(*

## Short summary
This class provides assert statements for pointers  

.. <legal notes>

legal notes
=================
| SPDX-FileCopyrightText: © 2022 ekvip automation GmbH <info@ekvip.de>
| SPDX-License-Identifier: Apache-2.0
| For details check: Apache-2.0_

.. _Apache-2.0: https://www.apache.org/licenses/LICENSE-2.0

.. </legal notes>



*)

{attribute 'reflection'}
FUNCTION_BLOCK PointerAssertions EXTENDS AbstractAssertion IMPLEMENTS IPointerAssertions
VAR
END_VAR

(*

## Short summary
This abstract property returns the class name of the concrete object, 
It's for debugging purpose

.. <legal notes>

legal notes
=================
| SPDX-FileCopyrightText: © 2022 ekvip automation GmbH <info@ekvip.de>
| SPDX-License-Identifier: Apache-2.0
| For details check: Apache-2.0_

.. _Apache-2.0: https://www.apache.org/licenses/LICENSE-2.0

.. </legal notes>

*)

PROPERTY className :CNM_AbstractObject.ClassName
GET
className := 'CNM_Assertor.PointerAssertions';
END_GET
END_PROPERTY

(*

## Short summary
This assertion method checks if pointer is aligned with register size.

.. <legal notes>

legal notes
=================
| SPDX-FileCopyrightText: © 2025 ekvip automation GmbH <info@ekvip.de>
| SPDX-License-Identifier: Apache-2.0
| For details check: Apache-2.0_

.. _Apache-2.0: https://www.apache.org/licenses/LICENSE-2.0

.. </legal notes>



*)

METHOD isAligned
VAR_INPUT
	(* memory address *)
	address		:PVOID;
	(* message if the assertion is false *)
	message		:AssertMessage;
END_VAR
VAR CONSTANT
	SIZE :PVOID := SIZEOF(__XWORD);
END_VAR
IF (address MOD SIZE > 0) THEN
	THIS^.assertionWasWrong(message, THIS^.getDebugInfo('isAligned'));
END_IF
END_METHOD

(*

## Short summary
This assertion method checks if pointer is aligned with DWord size.

.. <legal notes>

legal notes
=================
| SPDX-FileCopyrightText: © 2025 ekvip automation GmbH <info@ekvip.de>
| SPDX-License-Identifier: Apache-2.0
| For details check: Apache-2.0_

.. _Apache-2.0: https://www.apache.org/licenses/LICENSE-2.0

.. </legal notes>



*)

METHOD isDwordAligned
VAR_INPUT
	(* memory address *)
	address		:PVOID;
	(* message if the assertion is false *)
	message		:AssertMessage;
END_VAR
VAR CONSTANT
	SIZE :PVOID := SIZEOF(DWORD);
END_VAR
IF (address MOD SIZE > 0) THEN
	THIS^.assertionWasWrong(message, THIS^.getDebugInfo('isAligned'));
END_IF
END_METHOD

(*

## Short summary
This assertion method checks if ``address1`` and ``address2`` refer to the same address

.. <legal notes>

legal notes
=================
| SPDX-FileCopyrightText: © 2022 ekvip automation GmbH <info@ekvip.de>
| SPDX-License-Identifier: Apache-2.0
| For details check: Apache-2.0_

.. _Apache-2.0: https://www.apache.org/licenses/LICENSE-2.0

.. </legal notes>



*)

METHOD isEqualTo
VAR_INPUT
	(* memory address *)
	address1	:PVOID;
	(* memory address *)
	address2	:PVOID;
	(* message if the assertion is false *)
	message		:AssertMessage;
END_VAR
IF (address1 <> address2) THEN
	THIS^.assertionWasWrong(message, THIS^.getDebugInfo('isEqualTo'));
END_IF
END_METHOD

(*

## Short summary
This assertion method checks if pointer is aligned with Lword size.

.. <legal notes>

legal notes
=================
| SPDX-FileCopyrightText: © 2025 ekvip automation GmbH <info@ekvip.de>
| SPDX-License-Identifier: Apache-2.0
| For details check: Apache-2.0_

.. _Apache-2.0: https://www.apache.org/licenses/LICENSE-2.0

.. </legal notes>



*)

METHOD isLwordAligned
VAR_INPUT
	(* memory address *)
	address		:PVOID;
	(* message if the assertion is false *)
	message		:AssertMessage;
END_VAR
VAR CONSTANT
	SIZE :PVOID := SIZEOF(LWORD);
END_VAR
IF (address MOD SIZE > 0) THEN
	THIS^.assertionWasWrong(message, THIS^.getDebugInfo('isAligned'));
END_IF
END_METHOD

(*

## Short summary
This assertion method checks if ``address1`` and ``address2`` refer not to the same address

.. <legal notes>

legal notes
=================
| SPDX-FileCopyrightText: © 2022 ekvip automation GmbH <info@ekvip.de>
| SPDX-License-Identifier: Apache-2.0
| For details check: Apache-2.0_

.. _Apache-2.0: https://www.apache.org/licenses/LICENSE-2.0

.. </legal notes>



*)

METHOD isNotEqualTo
VAR_INPUT
	(* memory address *)
	address1	:PVOID;
	(* memory address *)
	address2	:PVOID;
	(* message if the assertion is false *)
	message		:AssertMessage;
END_VAR
IF (address1 = address2) THEN
	THIS^.assertionWasWrong(message, THIS^.getDebugInfo('isNotEqualTo'));
END_IF
END_METHOD

(*

## Short summary
This assertion method checks if pointer is not null

.. <legal notes>

legal notes
=================
| SPDX-FileCopyrightText: © 2022 ekvip automation GmbH <info@ekvip.de>
| SPDX-License-Identifier: Apache-2.0
| For details check: Apache-2.0_

.. _Apache-2.0: https://www.apache.org/licenses/LICENSE-2.0

.. </legal notes>



*)

METHOD isNotNull
VAR_INPUT
	(* memory address *)
	address	:PVOID;
	(* message if the assertion is false *)
	message	:AssertMessage;
END_VAR
IF (address = 0) THEN
	THIS^.assertionWasWrong(message, THIS^.getDebugInfo('isNotNull'));
END_IF
END_METHOD

(*

## Short summary
This assertion method checks if memory areas are overlapping

.. <legal notes>

legal notes
=================
| SPDX-FileCopyrightText: © 2022 ekvip automation GmbH <info@ekvip.de>
| SPDX-License-Identifier: Apache-2.0
| For details check: Apache-2.0_

.. _Apache-2.0: https://www.apache.org/licenses/LICENSE-2.0

.. </legal notes>



*)

METHOD isNotOverlapping
VAR_INPUT
	(* memory address *)
	address1	:PVOID;
	(* memory address *)
	address2	:PVOID;
	(*the size of the memory area identified by address1*)
	sizeInBytes1		:UDINT;
	(*the size of the memory area identified by address2*)
	sizeInBytes2		:UDINT;
	(* message if the assertion is false *)
	message		:AssertMessage;
END_VAR
IF 	(( 
		address1 = address2
	) OR_ELSE(
		//address1 + sizeInBytes1 < address1 is to protect overflows caused by the calculation address1 + sizeInBytes1
		(address1 < address2) AND_THEN ((address1 + sizeInBytes1 < address1) OR_ELSE ((address1 + sizeInBytes1) >= address2))
	) OR_ELSE (
		//address2 + sizeInBytes2 < address2 is to protect overflows caused by the calculation address2 + sizeInBytes2
		(address1 > address2) AND_THEN (((address2 + sizeInBytes2 < address2) OR_ELSE ((address2 + sizeInBytes2) >= address1)))
	)
) THEN
		THIS^.assertionWasWrong(message, THIS^.getDebugInfo('isNotOverlapping'));
END_IF
END_METHOD

(*

## Short summary
This assertion method checks if pointer is null

.. <legal notes>

legal notes
=================
| SPDX-FileCopyrightText: © 2022 ekvip automation GmbH <info@ekvip.de>
| SPDX-License-Identifier: Apache-2.0
| For details check: Apache-2.0_

.. _Apache-2.0: https://www.apache.org/licenses/LICENSE-2.0

.. </legal notes>



*)

METHOD isNull
VAR_INPUT
	(* memory address *)
	address	:PVOID;
	(* message if the assertion is false *)
	message	:AssertMessage;
END_VAR
IF (address <> 0) THEN
	THIS^.assertionWasWrong(message, THIS^.getDebugInfo('isNull'));
END_IF
END_METHOD

(*

## Short summary
This assertion method checks if memory areas are overlapping

.. <legal notes>

legal notes
=================
| SPDX-FileCopyrightText: © 2022 ekvip automation GmbH <info@ekvip.de>
| SPDX-License-Identifier: Apache-2.0
| For details check: Apache-2.0_

.. _Apache-2.0: https://www.apache.org/licenses/LICENSE-2.0

.. </legal notes>



*)

METHOD isOverlapping
VAR_INPUT
	(* memory address *)
	address1	:PVOID;
	(* memory address *)
	address2	:PVOID;
	(*the size of the memory area identified by address1*)
	sizeInBytes1		:UDINT;
	(*the size of the memory area identified by address2*)
	sizeInBytes2		:UDINT;
	(* message if the assertion is false *)
	message		:AssertMessage;
END_VAR
RETURN(address1 = address2);
IF ((
		(address1 < address2) AND_THEN ((address1 + sizeInBytes1) < address2)
	) OR_ELSE (
		(address1 > address2) AND_THEN ((address2 + sizeInBytes2) < address1)
	)
) THEN
	THIS^.assertionWasWrong(message, THIS^.getDebugInfo('isOverlapping'));
END_IF;
END_METHOD

(*

## Short summary
This assertion method checks if pointer is valid.
That means the pointer and size are not zero,
the pointer is in a valid area.

**Attention:** 
	Validity of the pointer will be proofed for 32 bit systems only.
	For other systems it's an optimistic estimate.

.. <legal notes>

legal notes
=================
| SPDX-FileCopyrightText: © 2022 ekvip automation GmbH <info@ekvip.de>
| SPDX-License-Identifier: Apache-2.0
| For details check: Apache-2.0_

.. _Apache-2.0: https://www.apache.org/licenses/LICENSE-2.0

.. </legal notes>



*)

METHOD isValid
VAR_INPUT
	(* memory address *)
	address		:PVOID;
	(* number of bytes *)
	sizeInBytes	:UDINT;
	(* message if the assertion is false *)
	message		:AssertMessage;
END_VAR
VAR
	{attribute 'displaymode':='hex'}
	stackAddress	:__XWORD;
	testPointer		:POINTER TO BYTE := NULL;
	testByte		:BYTE;
	exc				: __SYSTEM.ExceptionCode;
END_VAR
VAR CONSTANT
	{attribute 'displaymode':='hex'}
	NULL :__XWORD := 0;
	{attribute 'displaymode':='hex'}
	REGISTER_SIZE :UDINT := SIZEOF(__XWORD);
	(* 0x400000 is 4096kb and this is the max configurable stack size *)
	{attribute 'displaymode':='hex'}
	MAX_STACK_SIZE :__XWORD := 16#0040_0000;
END_VAR
stackAddress := ADR(stackAddress);
IF (
	(address = NULL) 
	OR_ELSE (sizeInBytes = NULL)
	//check for overflow
	OR_ELSE (address + sizeInBytes < address)
	OR_ELSE (
		(Tc2_System.F_CheckMemoryArea(pData := address, nSize := sizeInBytes) = Tc2_System.E_TcMemoryArea.Unknown)
		AND_THEN (address < ABS(stackAddress - MAX_STACK_SIZE))
	)
) THEN
	THIS^.assertionWasWrong(message, THIS^.getDebugInfo('isValid'));
ELSE
	testPointer := address;
	__TRY
		testByte := testPointer^;
	__CATCH(exc)
		THIS^.assertionWasWrong(message, THIS^.getDebugInfo('isValid'));
	__ENDTRY
END_IF
END_METHOD

(*

## Short summary
This assertion method checks if pointer is aligned with word size.

.. <legal notes>

legal notes
=================
| SPDX-FileCopyrightText: © 2025 ekvip automation GmbH <info@ekvip.de>
| SPDX-License-Identifier: Apache-2.0
| For details check: Apache-2.0_

.. _Apache-2.0: https://www.apache.org/licenses/LICENSE-2.0

.. </legal notes>



*)

METHOD isWordAligned
VAR_INPUT
	(* memory address *)
	address		:PVOID;
	(* message if the assertion is false *)
	message		:AssertMessage;
END_VAR
VAR CONSTANT
	SIZE :PVOID := SIZEOF(WORD);
END_VAR
IF (address MOD SIZE > 0) THEN
	THIS^.assertionWasWrong(message, THIS^.getDebugInfo('isAligned'));
END_IF
END_METHOD

(*

## Short summary
This assertion method checks if pointer refers to cnc area

.. <legal notes>

legal notes
=================
| SPDX-FileCopyrightText: © 2022 ekvip automation GmbH <info@ekvip.de>
| SPDX-License-Identifier: Apache-2.0
| For details check: Apache-2.0_

.. _Apache-2.0: https://www.apache.org/licenses/LICENSE-2.0

.. </legal notes>



*)

METHOD memoryAreaIsCnc
VAR_INPUT
	(* memory address *)
	address		:PVOID;
	(* number of bytes *)
	sizeInBytes	:UDINT;
	(* message if the assertion is false *)
	message		:AssertMessage;
END_VAR
IF (
	Tc2_System.F_CheckMemoryArea(
		pData := address,
		nSize := sizeInBytes
	) <> Tc2_System.E_TcMemoryArea.CNC
) THEN
	THIS^.assertionWasWrong(message, THIS^.getDebugInfo('memoryAreaIsCnc'));
END_IF
END_METHOD

(*

## Short summary
This assertion method checks if pointer refers to dynamic area

.. <legal notes>

legal notes
=================
| SPDX-FileCopyrightText: © 2022 ekvip automation GmbH <info@ekvip.de>
| SPDX-License-Identifier: Apache-2.0
| For details check: Apache-2.0_

.. _Apache-2.0: https://www.apache.org/licenses/LICENSE-2.0

.. </legal notes>



*)

METHOD memoryAreaIsDynamic
VAR_INPUT
	(* memory address *)
	address		:PVOID;
	(* number of bytes *)
	sizeInBytes	:UDINT;
	(* message if the assertion is false *)
	message		:AssertMessage;
END_VAR
IF (
	Tc2_System.F_CheckMemoryArea(
		pData := address,
		nSize := sizeInBytes
	) <> Tc2_System.E_TcMemoryArea.Dynamic
) THEN
	THIS^.assertionWasWrong(message, THIS^.getDebugInfo('memoryAreaIsDynamic'));
END_IF
END_METHOD

(*

## Short summary
This assertion method checks if pointer refers not to cnc area

.. <legal notes>

legal notes
=================
| SPDX-FileCopyrightText: © 2022 ekvip automation GmbH <info@ekvip.de>
| SPDX-License-Identifier: Apache-2.0
| For details check: Apache-2.0_

.. _Apache-2.0: https://www.apache.org/licenses/LICENSE-2.0

.. </legal notes>



*)

METHOD memoryAreaIsNotCnc
VAR_INPUT
	(* memory address *)
	address		:PVOID;
	(* number of bytes *)
	sizeInBytes	:UDINT;
	(* message if the assertion is false *)
	message		:AssertMessage;
END_VAR
IF (
	Tc2_System.F_CheckMemoryArea(
		pData := address,
		nSize := sizeInBytes
	) = Tc2_System.E_TcMemoryArea.CNC
) THEN
	THIS^.assertionWasWrong(message, THIS^.getDebugInfo('memoryAreaIsNotCnc'));
END_IF
END_METHOD

(*

## Short summary
This assertion method checks if pointer refers not to dynamic area

.. <legal notes>

legal notes
=================
| SPDX-FileCopyrightText: © 2022 ekvip automation GmbH <info@ekvip.de>
| SPDX-License-Identifier: Apache-2.0
| For details check: Apache-2.0_

.. _Apache-2.0: https://www.apache.org/licenses/LICENSE-2.0

.. </legal notes>



*)

METHOD memoryAreaIsNotDynamic
VAR_INPUT
	(* memory address *)
	address		:PVOID;
	(* number of bytes *)
	sizeInBytes	:UDINT;
	(* message if the assertion is false *)
	message		:AssertMessage;
END_VAR
IF (
	Tc2_System.F_CheckMemoryArea(
		pData := address,
		nSize := sizeInBytes
	) = Tc2_System.E_TcMemoryArea.Dynamic
) THEN
	THIS^.assertionWasWrong(message, THIS^.getDebugInfo('memoryAreaIsNotDynamic'));
END_IF
END_METHOD

(*

## Short summary
This assertion method checks if pointer refers not to static area

.. <legal notes>

legal notes
=================
| SPDX-FileCopyrightText: © 2022 ekvip automation GmbH <info@ekvip.de>
| SPDX-License-Identifier: Apache-2.0
| For details check: Apache-2.0_

.. _Apache-2.0: https://www.apache.org/licenses/LICENSE-2.0

.. </legal notes>



*)

METHOD memoryAreaIsNotStatic
VAR_INPUT
	(* memory address *)
	address		:PVOID;
	(* number of bytes *)
	sizeInBytes	:UDINT;
	(* message if the assertion is false *)
	message		:AssertMessage;
END_VAR
IF (
	Tc2_System.F_CheckMemoryArea(
		pData := address,
		nSize := sizeInBytes
	) = Tc2_System.E_TcMemoryArea.Static
) THEN
	THIS^.assertionWasWrong(message, THIS^.getDebugInfo('memoryAreaIsNotStatic'));
END_IF
END_METHOD

(*

## Short summary
This assertion method checks if pointer is not at memory area unknown

.. <legal notes>

legal notes
=================
| SPDX-FileCopyrightText: © 2022 ekvip automation GmbH <info@ekvip.de>
| SPDX-License-Identifier: Apache-2.0
| For details check: Apache-2.0_

.. _Apache-2.0: https://www.apache.org/licenses/LICENSE-2.0

.. </legal notes>



*)

METHOD memoryAreaIsNotUnkown
VAR_INPUT
	(* memory address *)
	address		:PVOID;
	(* number of bytes *)
	sizeInBytes	:UDINT;
	(* message if the assertion is false *)
	message		:AssertMessage;
END_VAR
IF (
	Tc2_System.F_CheckMemoryArea(
		pData := address,
		nSize := sizeInBytes
	) = Tc2_System.E_TcMemoryArea.Unknown
) THEN
	THIS^.assertionWasWrong(message, THIS^.getDebugInfo('memoryAreaIsNotUnkown'));
END_IF
END_METHOD

(*

## Short summary
This assertion method checks if pointer refers to static area

.. <legal notes>

legal notes
=================
| SPDX-FileCopyrightText: © 2022 ekvip automation GmbH <info@ekvip.de>
| SPDX-License-Identifier: Apache-2.0
| For details check: Apache-2.0_

.. _Apache-2.0: https://www.apache.org/licenses/LICENSE-2.0

.. </legal notes>



*)

METHOD memoryAreaIsStatic
VAR_INPUT
	(* memory address *)
	address		:PVOID;
	(* number of bytes *)
	sizeInBytes	:UDINT;
	(* message if the assertion is false *)
	message		:AssertMessage;
END_VAR
IF (
	Tc2_System.F_CheckMemoryArea(
		pData := address,
		nSize := sizeInBytes
	) <> Tc2_System.E_TcMemoryArea.Static
) THEN
	THIS^.assertionWasWrong(message, THIS^.getDebugInfo('memoryAreaIsStatic'));
END_IF
END_METHOD

(*

## Short summary
This assertion method checks if pointer refers not to an unknown area

.. <legal notes>

legal notes
=================
| SPDX-FileCopyrightText: © 2022 ekvip automation GmbH <info@ekvip.de>
| SPDX-License-Identifier: Apache-2.0
| For details check: Apache-2.0_

.. _Apache-2.0: https://www.apache.org/licenses/LICENSE-2.0

.. </legal notes>



*)

METHOD memoryAreaIsUnkown
VAR_INPUT
	(* memory address *)
	address		:PVOID;
	(* number of bytes *)
	sizeInBytes	:UDINT;
	(* message if the assertion is false *)
	message		:AssertMessage;
END_VAR
IF (
	Tc2_System.F_CheckMemoryArea(
		pData := address,
		nSize := sizeInBytes
	) <> Tc2_System.E_TcMemoryArea.Unknown
) THEN
	THIS^.assertionWasWrong(message, THIS^.getDebugInfo('memoryAreaIsUnkown'));
END_IF
END_METHOD

END_FUNCTION_BLOCK

(* stored: Version 1.1.0.1, ProductVersion 3.1.4026.11
   POU PointerAssertions: Id {26a0ce92-84f1-468d-9fe1-b917e2dfc179}, SpecialFunc None
   Property className: Id {3b83cf82-b6aa-426d-98fd-a94474afac43}
   Get Get: Id {f1923636-e634-46a8-895b-4b12e3a796c7}
   Method isAligned: Id {1049eedc-4d69-47ab-8f5c-cbf4b77c6ab7}
   Method isDwordAligned: Id {88ef15a2-62dd-4f6f-9697-be3bc959c47e}
   Method isEqualTo: Id {4a623468-b8c5-43af-af3a-ae6295531a4d}
   Method isLwordAligned: Id {9237bee0-2b96-4636-a6f3-1f054d045f39}
   Method isNotEqualTo: Id {54c4cb28-3f80-45df-ab44-82d97f69320a}
   Method isNotNull: Id {cd96bfa3-4cfb-41b2-b219-9b0c0a444683}
   Method isNotOverlapping: Id {41d2f5c9-34a5-4156-ac03-97141240756a}
   Method isNull: Id {544670de-ebfc-4740-85f3-1d121f65c90b}
   Method isOverlapping: Id {c9eb8344-714a-4db7-9fae-856fe8a9cf66}
   Method isValid: Id {4d85afcc-514f-4d0b-8ec9-b6734eb2854b}
   Method isWordAligned: Id {e7f88df0-f47b-468e-8785-347773d51856}
   Method memoryAreaIsCnc: Id {37f1e5c3-6d9b-406b-8449-a9977bd4d8c0}
   Method memoryAreaIsDynamic: Id {079c9284-01fe-40fe-b00c-97291b8dc55f}
   Method memoryAreaIsNotCnc: Id {20bbc746-04de-48d9-b522-d9702a64d96a}
   Method memoryAreaIsNotDynamic: Id {0395fb6f-7304-47d0-82a8-761411f58114}
   Method memoryAreaIsNotStatic: Id {329f55cf-3ab2-4189-8598-9d554de84359}
   Method memoryAreaIsNotUnkown: Id {95ccdc3f-cf8c-43ab-9fe0-2ac0cc87ccad}
   Method memoryAreaIsStatic: Id {7d735cd4-b968-41b3-87f1-2705a698bbd1}
   Method memoryAreaIsUnkown: Id {3731cdf9-9711-436d-97e4-2c40d31deba7} *)
